Staubli VAL3: start.pgx

program start()
begin
  // stop Cycle
  cycleStatus:bToStop=true
  watch(cycleStatus:bToStop==false,1)
end
